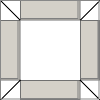
VISUALIZATION diaDataBox  // 100x100
VAR_IN_OUT
	iqBoxdata:structBoxData;
	
END_VAR
    Button (20,0 60x20), text list: 'textListTop', text index: iqBoxdata.topStatus
        OnMouseClick: toggle iqBoxdata.topStatusChange
    Button (0,20 20x60), text list: 'textListLeft', text index: iqBoxdata.leftStatus
        OnMouseClick: toggle iqBoxdata.leftStatusChange
    Button (80,20 20x60), text list: 'textListRight', text index: iqBoxdata.rightStatus
        OnMouseClick: toggle iqBoxdata.rightStatusChange
    Button (20,80 60x20), text list: 'textListBottom', text index: iqBoxdata.bottomStatus
        OnMouseClick: toggle iqBoxdata.bottomStatusChange
    Line (20,20) (0,0)
    Line (100,100) (80,80)
    Line (100,0) (80,20)
    Line (20,80) (0,100)
END_VISUALIZATION

(* stored: Version 1.1.0.1, ProductVersion 3.1.4024.11
   Visu diaDataBox: Id {7408d88e-96f1-0460-201c-08e7c14b3b44} *)
